ADAPTER Adapter1 (* Adapter Interface *)
  (* Standard: 61499-1 *)
  (* Version 0.0, 26/02/2026, Schneider Electric *)
  PACKAGE Hidryco.HidrycoLib;
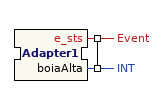
  EVENT_OUTPUT
    e_sts WITH boiaAlta;
  END_EVENT
  VAR_OUTPUT
    boiaAlta : INT;
  END_VAR
  SERVICE SOCKET/PLUG
    SEQUENCE request_confirm
      SOCKET.REQ(REQD) -> PLUG.REQ(REQD);
      PLUG.CNF(CNFD) -> SOCKET.CNF(CNFD);
    END_SEQUENCE
    SEQUENCE indication_response
      PLUG.IND(INDD) -> SOCKET.IND(INDD);
      SOCKET.RSP(RSPD) -> PLUG.RSP(RSPD);
    END_SEQUENCE
  END_SERVICE
END_ADAPTER
